Staubli VAL3: DELAY.pjx

--- DELAY.pjx ---
Parameters version=s7.5 stackSize=5000 millimeterUnit=true
Program file=find.pgx
Program file=get.pgx
Program file=getSize.pgx
Program file=getType.pgx
Program file=load.pgx
Program file=onEdit.pgx
Program file=onInsert.pgx
Program file=onProgEnd.pgx
Program file=onRun.pgx
Program file=onStart.pgx
Program file=onStop.pgx
Data file=DELAY.dtx
Library alias=use path=Disk://kernel/userPage/userPage.pjx
Library alias=cycleStatus path=Disk://cycleStatus/cycleStatus.pjx

--- onEdit.pgx ---
public program onEdit(string& x_sItem[])
  local num l_nX
  local num l_nY
  local num l_nDelay
  local bool l_bValide
begin
  // convert to a num
  l_bValide=true
  toNum(x_sItem,l_nDelay,l_bValide)
  // change the field
  call use:insertDialog("DELAY [Sec] ",l_nDelay,0,100)
  // give back
  if l_nDelay>0
    if round(l_nDelay)==l_nDelay
      x_sItem=toString("",l_nDelay)
    else
      x_sItem=toString(".2",l_nDelay)
    endIf
  endIf
end

--- onInsert.pgx ---
public program onInsert(string& x_sItem[])
  local num l_nDelay
begin
  cls()
  l_nDelay=0
  call use:insertDialog("DELAY [Sec] ",l_nDelay,0,100)
  // give back
  if l_nDelay>0
    if round(l_nDelay)==l_nDelay
      x_sItem=toString("",l_nDelay)
    else
      x_sItem=toString(".2",l_nDelay)
    endIf
  endIf
end

--- onRun.pgx ---
public program onRun(string& x_sItem[])
  local num l_nValue
  local bool l_bOk
begin
  //
  // convert to a num
  l_bOk=true
  toNum(x_sItem,l_nValue,l_bOk)
   // NB the robot will no STOP
  delay(l_nValue)
  //
end
